// TIA Portal V18 export
// export: Created 2026-06-06T00:00:00Z, ExportSetting WithDefaults
DATA_BLOCK "AI_Timers_PLC2"   // DB
TITLE = AI_Timers_PLC2
{ S7_Optimized_Access := 'TRUE' }
VERSION : 0.1
// Global DB containing all timers and PID instances
// stored: AutoNumber true, IsOnlyStoredInLoadMemory false, IsWriteProtectedInAS false
   VAR
      AI_Timer_Dosing_Bon3 : IEC_TIMER;
      AI_Timer_Tip_Bon3 : IEC_TIMER;
      AI_Timer_Dosing_Bon4 : IEC_TIMER;
      AI_Timer_Tip_Bon4 : IEC_TIMER;
      AI_Timer_Khuay_Bon3 : IEC_TIMER;
      AI_Timer_Khuay_Thuan_Bon4 : IEC_TIMER;
      AI_Timer_Khuay_Nghich_Bon4 : IEC_TIMER;
      AI_Timer_Thanh_Trung_Bon4 : IEC_TIMER;
      AI_Timer_DryRun_Bon4 : IEC_TIMER;
      AI_Timer_Heartbeat_PLC2 : IEC_TIMER;
   END_VAR
BEGIN
END_DATA_BLOCK
